PROGRAM DebugPro
VAR
    MC_MoveAbsolute_Axis: ARRAY[1..8] OF MC_MoveAbsolute ;
	MC_MoveAdditive_Axis: ARRAY[1..8] OF MC_MoveAdditive;
	MC_MoveRelative_Axis: array[1..8] of MC_MoveRelative;
	iDebug: INT;
	iDebugCyc: INT;
	tonDebug: Ton;
END_VAR

MC_MoveAbsolute_Axis[1](
	Axis:= arRealAxisAdmin[47].Axis, 
	Execute:= , 
	Position:= , 
	Velocity:= 10, 
	Acceleration:= 10, 
	Deceleration:= 10, 
	Jerk:= 10000, 
	BufferMode:= , 
	Options:= , 
	Done=> , 
	Busy=> , 
	Active=> , 
	CommandAborted=> , 
	Error=> , 
	ErrorID=> );

MC_MoveAbsolute_Axis[2](
	Axis:= arRealAxisAdmin[47].Axis, 
	Execute:= , 
	Position:= , 
	Velocity:= 100, 
	Acceleration:= 1000, 
	Deceleration:= 1000, 
	Jerk:= 10000, 
	BufferMode:= , 
	Options:= , 
	Done=> , 
	Busy=> , 
	Active=> , 
	CommandAborted=> , 
	Error=> , 
	ErrorID=> );	
	
MC_MoveAdditive_Axis[1](
	Axis:= arRealAxisAdmin[47].Axis, 
	Execute:= , 
	Distance:= , 
	Velocity:= 10, 
	Acceleration:= 100, 
	Deceleration:= 100, 
	Jerk:= 10000, 
	BufferMode:= , 
	Options:= , 
	Done=> , 
	Busy=> , 
	Active=> , 
	CommandAborted=> , 
	Error=> , 
	ErrorID=> );

MC_MoveAdditive_Axis[2](
	Axis:= arRealAxisAdmin[47].Axis, 
	Execute:= , 
	Distance:= , 
	Velocity:= 10, 
	Acceleration:= 100, 
	Deceleration:= 100, 
	Jerk:= 10000, 
	BufferMode:= , 
	Options:= , 
	Done=> , 
	Busy=> , 
	Active=> , 
	CommandAborted=> , 
	Error=> , 
	ErrorID=> );
		
MC_MoveRelative_Axis[1](
	Axis:= arRealAxisAdmin[47].Axis, 
	Execute:= , 
	Distance:= , 
	Velocity:= 10, 
	Acceleration:= 100, 
	Deceleration:= 100, 
	Jerk:= 10000, 
	BufferMode:= , 
	Options:= , 
	Done=> , 
	Busy=> , 
	Active=> , 
	CommandAborted=> , 
	Error=> , 
	ErrorID=> );	
	
MC_MoveRelative_Axis[2](
	Axis:= arRealAxisAdmin[47].Axis, 
	Execute:= , 
	Distance:= , 
	Velocity:= 10, 
	Acceleration:= 100, 
	Deceleration:= 100, 
	Jerk:= 10000, 
	BufferMode:= , 
	Options:= , 
	Done=> , 
	Busy=> , 
	Active=> , 
	CommandAborted=> , 
	Error=> , 
	ErrorID=> );	
	
CASE iDebug OF
	
10: MC_MoveAbsolute_Axis[1].Position:=100;
    MC_MoveAbsolute_Axis[1].Execute:=TRUE;
	IF MC_MoveAbsolute_Axis[1].Active THEN
	   MC_MoveAbsolute_Axis[1].Execute:=FALSE;
       iDebug:=20;
	END_IF
20:
    MC_MoveAbsolute_Axis[2].Position:=200;
    MC_MoveAbsolute_Axis[2].Execute:=TRUE;
	IF MC_MoveAbsolute_Axis[2].Active THEN
	   MC_MoveAbsolute_Axis[2].Execute:=FALSE;
	   iDebug:=iDebugCyc;
	END_IF
		
100: MC_MoveAdditive_Axis[1].Distance:=100;
    MC_MoveAdditive_Axis[1].Execute:=TRUE;
	IF MC_MoveAdditive_Axis[1].Active THEN
	   MC_MoveAdditive_Axis[1].Execute:=FALSE;
       iDebug:=200;
	END_IF
200:
    MC_MoveAdditive_Axis[2].Distance:=100;
    MC_MoveAdditive_Axis[2].Execute:=TRUE;
	IF MC_MoveAdditive_Axis[2].Active THEN
	   MC_MoveAdditive_Axis[2].Execute:=FALSE;
	   iDebug:=iDebugCyc;
	END_IF	
	
	
1000: MC_MoveRelative_Axis[1].Distance:=100;
    MC_MoveRelative_Axis[1].Execute:=TRUE;
	IF MC_MoveRelative_Axis[1].Active THEN
	   MC_MoveRelative_Axis[1].Execute:=FALSE;
       iDebug:=1100;
	END_IF
	
1100: 
     tonDebug(IN:= TRUE, PT:= T#1S, Q=> , ET=> );
	 IF tonDebug.Q THEN
		 tonDebug(IN:= FALSE, PT:= T#1S, Q=> , ET=> ); 
		 iDebug:=2000;
	 END_IF

	
2000:
    MC_MoveRelative_Axis[2].Distance:=100;
    MC_MoveRelative_Axis[2].Execute:=TRUE;
	IF MC_MoveRelative_Axis[2].Active THEN
	   MC_MoveRelative_Axis[2].Execute:=FALSE;
	   iDebug:=iDebugCyc;
	END_IF		
END_CASE

END_PROGRAM

(* stored: Version 1.1.0.1, ProductVersion 3.1.4024.6
   POU DebugPro: Id {c4a6157d-ce42-435e-9082-66b05b73bcc0}, SpecialFunc None *)
